FUNCTION_BLOCK diverter
  (* Standard: 61499-2 *)
  (* Version 0,1, 2015-00-16, Th?o, PC_THEO *)
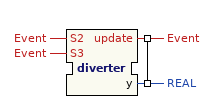
  EVENT_INPUT
    S2;
    S3;
  END_EVENT
  EVENT_OUTPUT
    update WITH y;
  END_EVENT
  VAR_OUTPUT
    y : REAL;
  END_VAR
  VAR
    theta : REAL;
  END_VAR
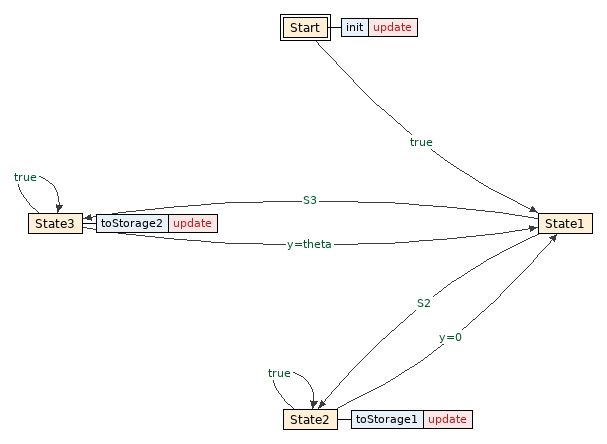
  EC_STATES
    Start : init -> update;
    State1;
    State2 : toStorage1 -> update;
    State3 : toStorage2 -> update;
  END_STATES
  EC_TRANSITIONS
    Start TO State1 := true;
    State1 TO State2 := S2;
    State1 TO State3 := S3;
    State2 TO State1 := y=0;
    State2 TO State2 := true;
    State3 TO State1 := y=theta;
    State3 TO State3 := true;
  END_TRANSITIONS
  ALGORITHM init IN C:
me->theta=6;
me->y=0;
  END_ALGORITHM
  ALGORITHM toStorage1 IN C:
if (me->y == 0){
	printf("diverter already in storage1, control error \n");
	exit(1);}

me->y=me->y-2;
printf("diverter, %f",me->y);
  END_ALGORITHM
  ALGORITHM toStorage2 IN C:
if (me->y == me->theta){
	printf("diverter already in storage2, control error \n");
	exit(1);}

if (me->y == me->theta){
	printf("diverter already in storage2, control error \n");
	exit(1);}

me->y=me->y+2;
printf("diverter, %f",me->y);
  END_ALGORITHM
END_FUNCTION_BLOCK
